ABB RAPID module: Singularidad_Munieca.mod

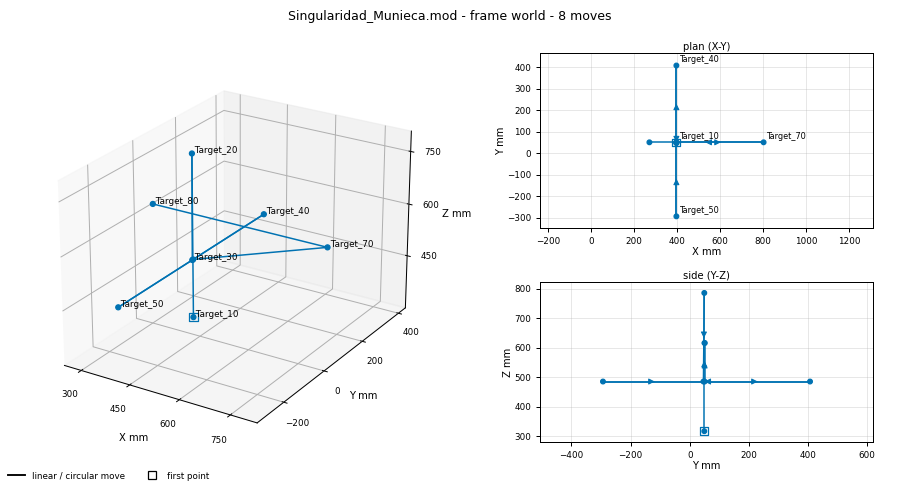
[picture p0: tool path of Singularidad_Munieca.mod in frame world, 8 of 8 moves have a stored position in this frame; points joined in program order, loops and branches not executed]
MODULE Module1
        CONST robtarget Target_10:=[[397.237379269,49.378335915,317.341657442],[0.500000149,-0.000000747,0.866025318,-0.000000248],[0,0,-1,1],[9E+09,9E+09,9E+09,9E+09,9E+09,9E+09]];
    CONST robtarget Target_20:=[[397.237401011,49.378342181,785.151469667],[0.500000129,-0.000000714,0.866025329,-0.000000203],[0,1,-2,1],[9E+09,9E+09,9E+09,9E+09,9E+09,9E+09]];
    CONST robtarget Target_30:=[[397.237400615,46.452570577,485.395596034],[0.500000124,-0.000000698,0.866025332,-0.0000002],[0,1,-1,1],[9E+09,9E+09,9E+09,9E+09,9E+09,9E+09]];
    CONST robtarget Target_40:=[[397.237407094,407.13958829,485.39559327],[0.500000134,-0.000000714,0.866025327,-0.000000239],[0,1,-1,1],[9E+09,9E+09,9E+09,9E+09,9E+09,9E+09]];
    CONST robtarget Target_50:=[[397.237392628,-293.472887343,485.395595719],[0.500000125,-0.000000729,0.866025331,-0.000000243],[-1,0,-2,0],[9E+09,9E+09,9E+09,9E+09,9E+09,9E+09]];
    CONST robtarget Target_60:=[[397.237393587,50.453069476,485.39558546],[0.500000114,-0.000000756,0.866025338,-0.000000264],[0,1,-1,1],[9E+09,9E+09,9E+09,9E+09,9E+09,9E+09]];
    CONST robtarget Target_70:=[[802.304016355,50.453065947,615.789609831],[0.500000141,-0.000000543,0.866025322,-0.000000186],[0,1,-2,1],[9E+09,9E+09,9E+09,9E+09,9E+09,9E+09]];
    CONST robtarget Target_80:=[[271.909522335,50.453072281,615.789590887],[0.500000145,-0.000000573,0.86602532,-0.000000214],[0,1,-2,1],[9E+09,9E+09,9E+09,9E+09,9E+09,9E+09]];
!***********************************************************
    !
    ! Module:  Module1
    !
    ! Description:
    !   <Insert description here>
    !
    ! Author: Ramiro
    !
    ! Version: 1.0
    !
    !***********************************************************


    !***********************************************************
    !
    ! Procedure main
    !
    !   This is the entry point of your program
    !
    !***********************************************************
    PROC main()
        Singularidad_Munieca;
    ENDPROC
    PROC Singularidad_Munieca()
        MoveJ Target_10,v1000,z100,tool0\WObj:=wobj0;
        MoveL Target_20,v1000,z100,tool0\WObj:=wobj0;
        MoveL Target_30,v1000,z100,tool0\WObj:=wobj0;
        MoveL Target_40,v1000,z100,tool0\WObj:=wobj0;
        MoveL Target_50,v1000,z100,tool0\WObj:=wobj0;
        MoveL Target_60,v1000,z100,tool0\WObj:=wobj0;
        MoveL Target_70,v1000,z100,tool0\WObj:=wobj0;
        MoveL Target_80,v1000,z100,tool0\WObj:=wobj0;
    ENDPROC
ENDMODULE
